ABB RobotStudio station: Test.rsstn

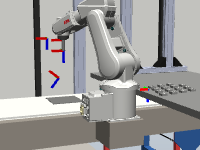
Station Station (saved by RobotStudio 6.7.7985.1011)
Controller MTRN4230, task T_ROB1: task frame (RAPID world) sits at (2935, -1760, 590) mm in the station
Controller MTRN4230
  mechanical unit ROB_1: IRB120_3_58__01, 6 joints, base frame (0, 0, 0) mm
Layout (positions relative to the parent item):
  - IRB120_3_58__01 [mechanism, from Robots\IRB120_3_58_G_01.rslib] at (2935, -1760, 590) mm; joint values [2.0779, 0.4446, -0.0557, 0, 1.1819, 2.0779] (rad or m)
  - ROBOTROOM [part] at (3020, -2855, 1950) mm, rotated rx 90 ry 0 rz 0 deg
  - ConvBox [part] at (29.42, 180.2, -38.47) mm
  - SmartComponent_1 [smart component]
    - CollisionSensor [smart component, from Components\CollisionSensor.rslib]
        properties: Object1=(none); Object2=(none); NearMiss=0; Part1=(none); Part2=(none); CollisionType=0
  - Attacher [smart component, from Components\Attacher.rslib]
      properties: Parent=MyNewTool; Flange=0; Child=letterblock_3; Mount=false; Offset=[0 0 0]; Orientation=[0 0 0]
  - Detacher [smart component, from Components\Detacher.rslib]
      properties: Child=letterblock_3; KeepPosition=true
  - Group_1 [graphiccomponentgroup] at (0, 0, 0) mm
    - letterblock_2 [part] at (3128, -1904, 730) mm, rotated rx 90 ry 0 rz 180 deg
    - letterblock_3 [part] at (3146, -1832, 730) mm, rotated rx 90 ry 0 rz 180 deg
    - letterblock_4 [part] at (3164, -1760, 730) mm, rotated rx 90 ry 0 rz 180 deg
    - letterblock_5 [part] at (3182, -1688, 730) mm, rotated rx 90 ry 0 rz 180 deg
    - letterblock_6 [part] at (3200, -1886, 730) mm, rotated rx 90 ry 0 rz 180 deg
    - letterblock_7 [part] at (3218, -1814, 730) mm, rotated rx 90 ry 0 rz 180 deg
    - letterblock_8 [part] at (3236, -1742, 730) mm, rotated rx 90 ry 0 rz 180 deg
    - letterblock_9 [part] at (3254, -1670, 730) mm, rotated rx 90 ry 0 rz 180 deg
    - letterblock_10 [part] at (3272, -1868, 730) mm, rotated rx 90 ry 0 rz 180 deg
    - letterblock_11 [part] at (3290, -1796, 730) mm, rotated rx 90 ry 0 rz 180 deg
    - letterblock_12 [part] at (3308, -1724, 730) mm, rotated rx 90 ry 0 rz 180 deg
    - letterblock_13 [part] at (3326, -1652, 730) mm, rotated rx 90 ry 0 rz 180 deg
    - letterblock_14 [part] at (3344, -1850, 730) mm, rotated rx 90 ry 0 rz 180 deg
    - letterblock_15 [part] at (3362, -1778, 730) mm, rotated rx 90 ry 0 rz 180 deg
    - letterblock_16 [part] at (3380, -1706, 730) mm, rotated rx 90 ry 0 rz 180 deg
    - letterblock_17 [part] at (-416, 441, 197) mm
  - CollisionSensor [smart component, from Components\CollisionSensor.rslib]
      properties: Object1=MyNewTool; Object2=Group_1; NearMiss=0.01; Part1=Endeffector; Part2=letterblock_3; CollisionType=2
  - MyNewTool [mechanism] at (2730, -1391, 1002) mm, rotated rx 180 ry 0 rz 180 deg
      TCP MyNewTool at (36.7, 266.44, 0) mm
      links: Endeffector
  - CollisionSensor_2 [smart component, from Components\CollisionSensor.rslib]
      properties: Object1=ROBOTROOM; Object2=Group_1; NearMiss=0.01; Part1=ROBOTROOM; Part2=letterblock_17; CollisionType=2
  - LogicGate [smart component, from Components\LogicGate.rslib]
      properties: Operator=NOT; Delay=0
  - coords [frame] at (2935, -1760, 590) mm
Attachment: MyNewTool is attached to IRB120_3_58__01 / Link6
Attachment: letterblock_17 is attached to MyNewTool / Endeffector
EventTableEntry 1093: Group=, Trigger=EventTableTriggerCollision 1094, Actions=[EventTableActionAttach 1209], Comment=, ActivationMode=2, Cyclic=false
EventTableTriggerCollision 1094: CollisionSet=CollisionSet_1 1099, EventType=1
EventTableEntry 1096: Group=, Trigger=EventTableTriggerCollision 1097, Actions=[EventTableActionDetach 1202], Comment=, ActivationMode=2, Cyclic=false
EventTableTriggerCollision 1097: CollisionSet=CollisionSet_5 1216, EventType=1
Collision set CollisionSet_1: MyNewTool against letterblock_2, near miss 0.005 m
Collision set CollisionSet_2: MyNewTool against letterblock_6, near miss 0.005 m
EventTableActionDetach 1202: AttachmentParent=MyNewTool 1195, AttachmentChild=letterblock_2 1116
EventTableActionAttach 1209: AttachmentParent=MyNewTool 1195, AttachmentChild=letterblock_2 1116, MountObject=false, Offset=[X=1, Y=0, Z=0, W=0, X=0, Y=1, Z=0, W=0, X=0, Y=0, Z=1, W=0, X=0, Y=0, Z=0, W=1], FlangeIndext=0, FindNearest=false
EventTableEntry 1210: Group=, Trigger=EventTableTriggerCollision 1211, Actions=[EventTableActionAttach 1212], Comment=, ActivationMode=2, Cyclic=false
EventTableTriggerCollision 1211: CollisionSet=CollisionSet_2 1100, EventType=1
EventTableActionAttach 1212: AttachmentParent=MyNewTool 1195, AttachmentChild=letterblock_6 1124, MountObject=false, Offset=[X=1, Y=0, Z=0, W=0, X=0, Y=1, Z=0, W=0, X=0, Y=0, Z=1, W=0, X=0, Y=0, Z=0, W=1], FlangeIndext=0, FindNearest=false
EventTableEntry 1213: Group=, Trigger=EventTableTriggerCollision 1214, Actions=[EventTableActionDetach 1215], Comment=, ActivationMode=2, Cyclic=false
EventTableTriggerCollision 1214: CollisionSet=CollisionSet_6 1217, EventType=1
EventTableActionDetach 1215: AttachmentParent=MyNewTool 1195, AttachmentChild=letterblock_6 1124
Collision set CollisionSet_5: letterblock_2 against ConvBox, near miss 0 m
Collision set CollisionSet_6: letterblock_6 against ConvBox, near miss 0 m
Station signals: DI DI10_1
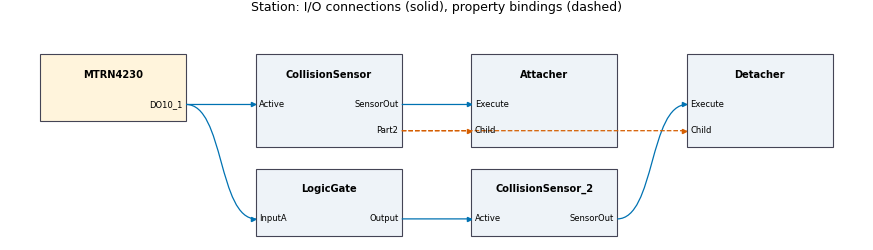
Station logic (signal -> signal, property => property):
  CollisionSensor.SensorOut -> Attacher.Execute
  CollisionSensor_2.SensorOut -> Detacher.Execute
  MTRN4230.DO10_1 -> CollisionSensor.Active
  MTRN4230.DO10_1 -> LogicGate.InputA
  LogicGate.Output -> CollisionSensor_2.Active
  CollisionSensor.Part2 => Detacher.Child
  CollisionSensor.Part2 => Attacher.Child
Targets, tools, work objects and paths stored in the station, written as RAPID:
! task T_ROB1
MODULE MTRN4230_Move_Sample
  PROC MoveJSample()
    MoveJ pTableHome,v100,fine,tSCup;
  ENDPROC
  PROC MoveLSample()
    MoveL Offs(pTableHome, 0, 0, 100),v100,fine,tSCup;
  ENDPROC
  PROC MainMove()
    MoveJSample;
    MoveLSample;
  ENDPROC
ENDMODULE

! task T_ROB1
MODULE MTRN4230_IO_Sample
  PROC MainIO()
    TurnVacOn;
    WaitTime 2;
    TurnVacOff;
    TurnConOnSafely;
    WaitTime 2;
    TurnConOff;
  ENDPROC
  PROC TurnVacOff()
    SetDO DO10_1,0;
  ENDPROC
  PROC TurnConOff()
    SetDO DO10_3,0;
  ENDPROC
  PROC TurnVacOn()
    SetDO DO10_1,1;
  ENDPROC
  PROC TurnConOnSafely()
    SetDO DO10_3,1;
    SetDO DO10_3,0;
  ENDPROC
ENDMODULE

! task T_ROB1
MODULE MTRN_Rob_Data
  CONST robtarget pTableHome:=[[175,0,147],[0,0,1,0],[0,0,0,0],[9E+09,9E+09,9E+09,9E+09,9E+09,9E+09]];
  PERS tooldata tSCup:=[TRUE,[[0,0,65],[1,0,0,0]],[0.5,[0,0,20],[1,0,0,0],0,0,0]];
ENDMODULE

! task T_ROB1
MODULE CalibData
  PERS tooldata MyTool:=[TRUE,[[31.792631019,0,229.638935148],[0.945518576,0,0.325568154,0]],[1,[0,0,1],[1,0,0,0],0,0,0]];
  PERS tooldata MyNewTool:=[TRUE,[[36.697,266.435,0],[1,0,0,0]],[0.2,[0,0,1],[1,0,0,0],0,0,0]];
ENDMODULE

